PROGRAM MAIN
VAR
END_VAR

SFC();

END_PROGRAM

(* stored: Version 1.1.0.1, ProductVersion 3.1.4024.12
   POU MAIN: Id {87855124-4e36-45cb-89d0-ae7ecdb3dc67}, SpecialFunc None *)
